FUNCTION_BLOCK sfc_TCPServer
VAR_INPUT
	sLocalHost: T_IPv4Addr;
	nLocalPort: UDINT;
	bStartCommunication : BOOL;
END_VAR
VAR_OUTPUT
	bConnected: BOOL;
	eCommand : E_CommandList;
	sSendData: STRING(255);
	bBusy: BOOL;	
	bError: BOOL;
	nErrorID: UDINT;
END_VAR
VAR
	
	// State Vars
	iState				: INT;
	xInit				: R_TRIG;
	xOpenSocket			: R_TRIG;
	xError0				: R_TRIG;
	xError1				: R_TRIG;
	xError2				: R_TRIG;
	xError3				: R_TRIG;
	xError4				: R_TRIG;
	xError5				: R_TRIG;
	xAcceptConnection	: R_TRIG;
	xReceiveData		: R_TRIG;
	xParseData			: R_TRIG;
	xClearBuff			: R_TRIG;
	xSendData			: R_TRIG;
	xErrHandle			: R_TRIG;
	xPreClose			: R_TRIG;
	xCloseSocket		: R_TRIG;
	xReset				: R_TRIG;
	
	hListener: T_HSOCKET;
	hSocket: T_HSOCKET;
	fbSocketAccept: FB_SocketAccept;
	fbSocketListen: FB_SocketListen;
	fbLinkStatus: FB_IpAdapterGetLinkStatus;
	fbSocketReceive: FB_SocketReceive;
	fbSocketClose: FB_SocketClose;
	fbSocketCloseAll: FB_SocketCloseAll;
	fbSocketSend: FB_SocketSend;
	bAcceptExecute: BOOL;
	bAccepted: BOOL;
	bLinkError: BOOL;
	bStatusExecute: BOOL;
	
	ReceiveCounter: UDINT;
	sReadData: STRING(255);
	
	bSendTrigger: BOOL;
	
	// String Parse
    nLength : INT;
	sCommand : STRING(255);
	sTail	 : STRING(255);
	sBuff    : STRING(255);
	// Server Response
	bReturn : BOOL;
END_VAR

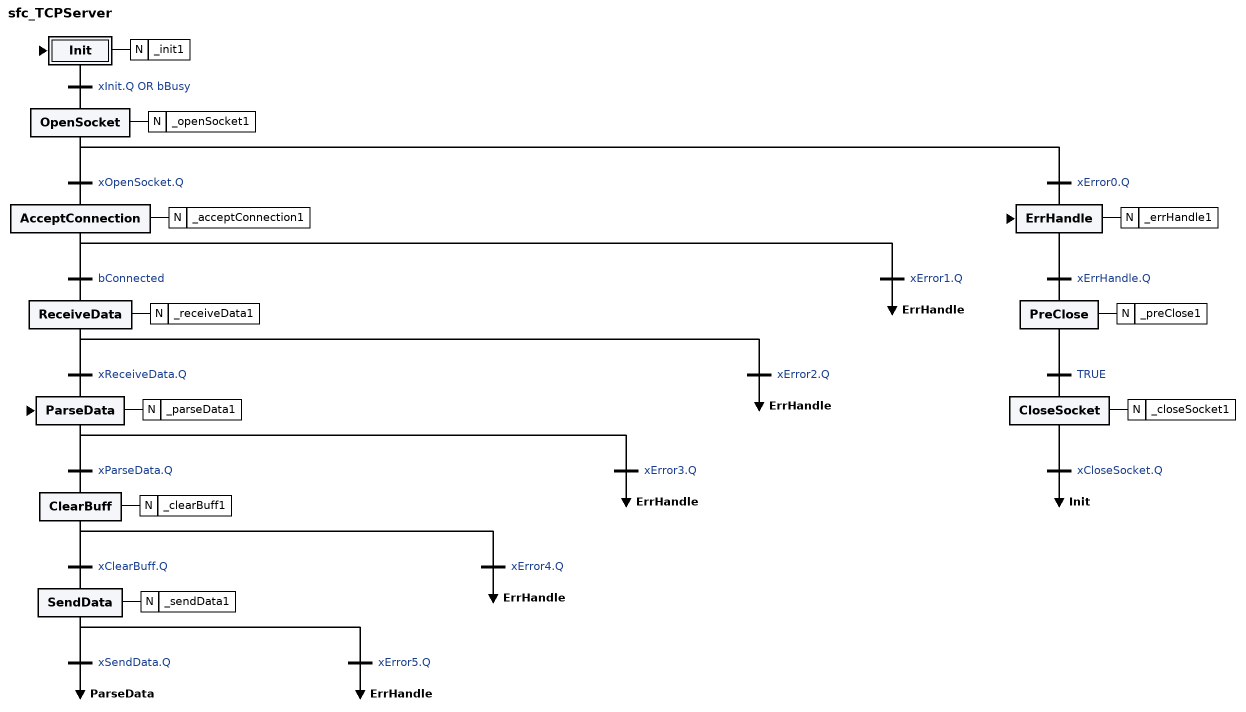
INITIAL_STEP Init:
    _init1(N);
END_STEP
TRANSITION FROM Init TO OpenSocket
    := xInit.Q OR bBusy;
END_TRANSITION
STEP OpenSocket:
    _openSocket1(N);
END_STEP
TRANSITION FROM OpenSocket TO AcceptConnection
    := xOpenSocket.Q;
END_TRANSITION
TRANSITION FROM OpenSocket TO ErrHandle
    := xError0.Q;
END_TRANSITION
STEP ErrHandle:
    _errHandle1(N);
END_STEP
TRANSITION FROM ErrHandle TO PreClose
    := xErrHandle.Q;
END_TRANSITION
STEP PreClose:
    _preClose1(N);
END_STEP
TRANSITION FROM PreClose TO CloseSocket
    := TRUE;
END_TRANSITION
STEP CloseSocket:
    _closeSocket1(N);
END_STEP
TRANSITION FROM CloseSocket TO Init
    := xCloseSocket.Q;
END_TRANSITION
STEP AcceptConnection:
    _acceptConnection1(N);
END_STEP
TRANSITION FROM AcceptConnection TO ReceiveData
    := bConnected;
END_TRANSITION
TRANSITION FROM AcceptConnection TO ErrHandle
    := xError1.Q;
END_TRANSITION
STEP ReceiveData:
    _receiveData1(N);
END_STEP
TRANSITION FROM ReceiveData TO ParseData
    := xReceiveData.Q;
END_TRANSITION
TRANSITION FROM ReceiveData TO ErrHandle
    := xError2.Q;
END_TRANSITION
STEP ParseData:
    _parseData1(N);
END_STEP
TRANSITION FROM ParseData TO ClearBuff
    := xParseData.Q;
END_TRANSITION
TRANSITION FROM ParseData TO ErrHandle
    := xError3.Q;
END_TRANSITION
STEP ClearBuff:
    _clearBuff1(N);
END_STEP
TRANSITION FROM ClearBuff TO SendData
    := xClearBuff.Q;
END_TRANSITION
TRANSITION FROM ClearBuff TO ErrHandle
    := xError4.Q;
END_TRANSITION
STEP SendData:
    _sendData1(N);
END_STEP
TRANSITION FROM SendData TO ParseData
    := xSendData.Q;
END_TRANSITION
TRANSITION FROM SendData TO ErrHandle
    := xError5.Q;
END_TRANSITION

ACTION _acceptConnection1:
fbSocketAccept(
	sSrvNetId:= '',         
	hListener:= hListener,                                           // Handle of Listener Socket
	bExecute:= TRUE, 
	tTimeout:= T#4S, 
	bAccepted=> bAccepted, 
	bBusy=> , 
	bError=> bError, 
	nErrId=> nErrorID,
	hSocket=> hSocket);                                              // Connection Handle

xAcceptConnection(CLK:=(hSocket.handle <> 0));
IF NOT fbSocketAccept.bBusy THEN
	fbSocketAccept(bExecute := FALSE);
END_IF

fbLinkStatus(sSrvNetId:= '',
				   sLocalHost := sLocalHost,
				   bExecute := bStatusExecute,
				   tTimeout := T#4S,
				   bLinkError => bLinkError);
	   

IF hSocket.handle <> 0 THEN
	bConnected := TRUE;									
END_IF
xError1(CLK:=bError);
END_ACTION

ACTION _clearBuff1:

// Clear ReceiveBuffer after processing
xClearBuff(CLK:= (memset(ADR(sReadData), 0, SIZEOF(sReadData))>0));
(*memset(ADR(sServerEcho), 0, SIZEOF(sServerEcho));
memset(ADR(sEchoFooter), 0, SIZEOF(sEchoFooter));
memset(ADR(sEchoHeader), 0, SIZEOF(sEchoHeader));*)        

{'warning': Need TO ADD conditional here}
END_ACTION

ACTION _closeSocket1:

fbSocketClose(
	sSrvNetId:= '', 
	hSocket:= hSocket, 
	bExecute:= TRUE, 
	tTimeout:= T#4S, 
	bBusy=> , 
	bError=> bError, 
	nErrId=> nErrorID);


IF NOT (fbSocketClose.bBusy) OR fbSocketClose.bError THEN
	hSocket.handle := 0;    
	bConnected := FALSE;
END_IF
xCloseSocket(CLK:=(NOT (fbSocketClose.bBusy) OR fbSocketClose.bError));
END_ACTION

ACTION _errHandle1:

// Error Handling    
fbSocketClose(                                                        // Close Listener-Socket
	sSrvNetId:= '', 
	hSocket:= hListener, 
	bExecute:= TRUE, 
	tTimeout:= T#4S, 
	bBusy=> , 
	bError=> bError, 
	nErrId=> nErrorID);        

IF (NOT fbSocketClose.bBusy) OR fbSocketClose.bError THEN
	hListener.handle := 0;
END_IF
xErrHandle(CLK:=((NOT fbSocketClose.bBusy) OR fbSocketClose.bError));
END_ACTION

ACTION _init1:
xInit(CLK:=bStartCommunication);
IF bStartCommunication = TRUE THEN
	fbSocketListen(bExecute := FALSE);
	fbSocketAccept(bExecute := FALSE);
	fbSocketCloseAll(bExecute := FALSE);
	fbSocketClose(bExecute:= FALSE);
	bConnected := FALSE;
	bBusy := TRUE;
	

ELSE
	bBusy := FALSE;
END_IF
END_ACTION

ACTION _openSocket1:

// Open Listener-Socket
fbSocketListen(
	sSrvNetId:= '',                                                 // Local NetID
	sLocalHost:= sLocalHost,                                         // Local IP
	nLocalPort:= nLocalPort,                                         // Local Port
	bExecute:= TRUE, 
	tTimeout:= T#4S, 
	bBusy=> , 
	bError=> bError, 
	nErrId=> nErrorID,
	hListener=> hListener);                                          // Handle of Listener Socket
	
xOpenSocket(CLK:=hListener.handle <> 0);
xError0(CLK:= bError);
END_ACTION

METHOD _ParseCommand : INT
VAR_INPUT
END_VAR
// Step 1: Parse out the command and tail
nLength := LEN(sReadData);
sTail := CONCAT('$0D','$0A');
IF nLength > 2 THEN
    sCommand := LEFT(sReadData, nLength - 2);  // Remove CR LF
END_IF

// Step 2: Command matching
IF sCommand = 'LIST' THEN
    _ParseCommand := E_CommandList.LIST;
ELSIF sCommand = 'HOM' THEN
    _ParseCommand := E_CommandList.HOM;
ELSIF sCommand = 'SCAN' THEN
    _ParseCommand := E_CommandList.SCAN;
ELSIF sCommand = 'MTP' THEN
    _ParseCommand := E_CommandList.MTP;
ELSIF sCommand = 'MOVR' THEN
    _ParseCommand := E_CommandList.MOVR;
ELSIF sCommand = 'MOVA' THEN
    _ParseCommand := E_CommandList.MOVA;
ELSIF sCommand = 'STAT' THEN
    _ParseCommand := E_CommandList.STAT;
ELSIF sCommand = 'CALIB' THEN
    _ParseCommand := E_CommandList.CALIB;
ELSIF sCommand = 'PARAM' THEN
    _ParseCommand := E_CommandList.PARAM;
ELSE
    _ParseCommand := E_CommandList.ERR;  // Unknown command
END_IF
END_METHOD

ACTION _parseData1:

// Parse Data
	eCommand := _ParseCommand();
	CASE eCommand OF
		E_CommandList.LIST:
			// List out available command
			bReturn := _SendServerResponse('LIST, HOM, SCAN, MTP, MOVR, MOVA, STAT, CALIB, PARAM');
		E_CommandList.HOM:
			// Home
			bReturn := _SendServerResponse('HOM');
		E_CommandList.SCAN:
			// Scan
			bReturn := _SendServerResponse('SCAN');
		E_CommandList.MTP:
			// Move to Pod
			bReturn := _SendServerResponse('MTP');
		E_CommandList.MOVR:
			// Move Relative
			bReturn := _SendServerResponse('MOVR');
		E_CommandList.MOVA:
			// Move Absolute
			bReturn := _SendServerResponse('MOVA');
		E_CommandList.STAT:
			// Machine Status
			bReturn := _SendServerResponse('STAT');
		E_CommandList.CALIB:
			// Machine Calibration Scan
			bReturn := _SendServerResponse('CALIB');
		E_CommandList.PARAM:
			// Set Parameters Mode
			bReturn := _SendServerResponse('PARAM');
		E_CommandList.ERR:
			// Command error
			bReturn := _SendServerResponse('ERR');
	END_CASE
	xParseData(CLK:= (eCommand <> E_CommandList.NULL));
	//_ParseData := TRUE;
	{'warning': Need to add conditional here to prevent race condition}
END_ACTION

ACTION _preClose1:

fbSocketClose(bExecute := FALSE);
END_ACTION

ACTION _receiveData1:

// Receive Data
fbSocketReceive(                                                     // Check cyclically for new client data 
	sSrvNetId:= '', 
	hSocket:= hSocket, 
	cbLen:= SIZEOF(sReadData), 
	pDest:= ADR(sReadData), 
	bExecute:= TRUE,                                                 
	tTimeout:= T#4S, 
	bBusy=> , 
	bError=> bError, 
	nErrId=> nErrorID,
	nRecBytes=> );

IF NOT fbSocketReceive.bBusy THEN
	fbSocketReceive(bExecute := FALSE);
	
	IF fbSocketReceive.nRecBytes <> 0 THEN                            // Switch to send-state when data are received
		fbSocketSend(bExecute := FALSE);             
		
		
	END_IF
END_IF
xReceiveData(CLK := fbSocketReceive.nRecBytes <> 0);
xError2(CLK:=(fbSocketReceive.bError OR (NOT bStartCommunication)));
// Close connection when error is occurring or trigger is set
END_ACTION

ACTION _sendData1:

// Send Data
fbSocketSend(                                                        // Send Data to client
	sSrvNetId:= '', 
	hSocket:= hSocket, 
	cbLen:= SIZEOF(sSendData), 
	pSrc:= ADR(sSendData),
	bExecute:= TRUE, 
	tTimeout:= T#3S, 
	bBusy=> , 
	bError=> bError, 
	nErrId=> nErrorID);    

IF NOT fbSocketSend.bBusy THEN                                        // Switch back to receiving state after sending
	memset(ADR(sSendData), 0, SIZEOF(sSendData));
	eCommand := E_CommandList.NULL;
END_IF
xSendData(CLK:=NOT fbSocketSend.bBusy);
xError5(CLK:=fbSocketSend.bError);
END_ACTION

METHOD _SendServerResponse : BOOL
VAR_INPUT
	sResponseText : STRING(255);
END_VAR
VAR
    sCRLF : STRING := '$0D$0A';
    sFinalResponse : STRING(255);
    nResponseSize : INT;
END_VAR
// Build the full response
sFinalResponse := CONCAT(sResponseText, sCRLF);

// Copy response to send buffer
nResponseSize := LEN(sFinalResponse);
memcpy(ADR(sSendData), ADR(sFinalResponse), nResponseSize);

// Null-terminate
sSendData[nResponseSize] := 0;
END_METHOD

METHOD transit : BOOL
VAR_INPUT
    xCondition : BOOL;  // Input condition for transition
    xReset : BOOL;      // Input to reset the condition
END_VAR
VAR_OUTPUT
    bTransitioned : BOOL;  // Output TRUE if transition occurs
END_VAR
VAR
    rTrig : R_TRIG;  // Rising edge detector
END_VAR
// Initialize default output
bTransitioned := FALSE;

// Perform rising edge detection on the input condition
rTrig(CLK := xCondition);

// If a rising edge is detected, it means a transition is triggered
IF rTrig.Q THEN
    bTransitioned := TRUE;  // Transition has occurred
END_IF

// Reset the condition if requested to close the transition
IF xReset THEN
    bTransitioned := FALSE;  // Clear transition flag
END_IF

// Return the result of the transition
transit := bTransitioned;
END_METHOD

END_FUNCTION_BLOCK

(* stored: Version 1.1.0.1, ProductVersion 3.1.4024.12
   POU sfc_TCPServer: Id {3ce36fc9-1762-452e-b306-7c91704ff748}, SpecialFunc None
   Action _acceptConnection1: Id {2ca79605-7a1b-4ee7-a761-85ebdc83a504}
   Action _clearBuff1: Id {fb522c91-6d82-475d-acef-b1167eec1f56}
   Action _closeSocket1: Id {718ea137-5f3e-4e6d-a244-ed7a23c400d5}
   Action _errHandle1: Id {7ebc9ab9-a2a9-4570-9b6d-ac70357a9d8e}
   Action _init1: Id {45a8aa93-8427-4d8d-8c06-ae1a80c790c7}
   Action _openSocket1: Id {ebb0ace3-a124-47f5-872a-1adf6feaf211}
   Method _ParseCommand: Id {909b6975-3b64-41ec-8d2a-7a71cb0e7f7f}
   Action _parseData1: Id {900c71ae-ea2a-4e32-832d-f11033606a82}
   Action _preClose1: Id {9c3f33af-cc26-4e6d-ac7d-1e3bbdfcd2a1}
   Action _receiveData1: Id {4c615df4-7da8-4cc2-bc13-b52f8658a21f}
   Action _sendData1: Id {bbc024a4-2f3b-49f9-9a47-4f82df3ad587}
   Method _SendServerResponse: Id {36750eef-660b-45b4-9ade-e9f03184808b}
   Method transit: Id {d850f324-7a04-4d44-b25f-dfbda85d7086} *)
